FUNCTION_BLOCK FB_CommandChangeHold EXTENDS FB_CommandChange IMPLEMENTS ITF_CommandChange
VAR

END_VAR

METHOD Execute : BOOL
VAR_INPUT
END_VAR
END_METHOD

END_FUNCTION_BLOCK

(* stored: Version 1.1.0.1
   POU FB_CommandChangeHold: Id {247ccda2-a7e4-023b-09df-f50757b37973}, SpecialFunc None
   Method Execute: Id {8068ef73-9267-022e-0e89-310894ff9a6d} *)
